FUNCTION_BLOCK FB_SendingData

END_FUNCTION_BLOCK

(* stored: Version 1.1.0.1, ProductVersion 3.1.4024.16
   POU FB_SendingData: Id {ad5a99aa-9b16-4636-8c02-6ad35f0f0b60}, SpecialFunc None *)
